{attribute 'OPC.UA.DA.StructuredType' := '1'}
TYPE ST_ActiveStorageSystemSetParameters :
STRUCT
	bLoadingAlgorithm: BOOL;
	bLoadingManual : BOOL;
END_STRUCT
END_TYPE

(* stored: Version 1.1.0.1, ProductVersion 3.1.4024.10
   DUT ST_ActiveStorageSystemSetParameters: Id {c086b274-3cd2-4559-bd3e-7d410ecfc5b1} *)
